ABB RobotStudio station: AGS01Tool.rspag

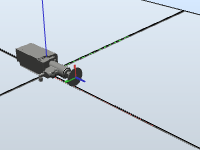
Station Station (saved by RobotStudio 6.4.7206.1027)
Layout (positions relative to the parent item):
  - AGS01Tool [mechanism, from abb\AGS01Tool.rslib] at (0, 0, 0) mm
  - AGS01Tcp [frame] at (154.8, 0, 42) mm, rotated rx 0 ry -90 rz -180 deg
